// TIA Portal V20 export
DATA_BLOCK "Instance_FB_Recive_Water_Fountain_From_Rework_DB"   // DB105
// stored: AutoNumber false, InstanceOfName FB_Recive_Water_Fountain_From_Rework, InstanceOfType FB
"FB_Recive_Water_Fountain_From_Rework"
   // VAR_INPUT
   //    Emergency_Stop_Release : Bool;
   //    Start : Bool;
   //    Sensor_Water_Fountain_Before_Entrace_Functional_Test_Spinner_Conveyor_Belt : Bool;
   //    Sensor_Water_Fountain_Entrace_Functional_Test_Spinner_Conveyor_Belt : Bool;
   //    Sensor_Spinner_Entrace_Functional_Test_Position_Withdrawn : Bool;
   //    Sensor_Spinner_Entrace_Functional_Test_Position_Advanced : Bool;
   //    Sensor_Water_Fountain_Entrace_Functional_Test_After_Spinner_Conveyor_Belt : Bool;
   //    Sensor_Water_Fountain_Geting_Exit_Rework_Conveyor_Belt : Bool;
   //    Button_Water_Fountain_Get_Exit_Rework_Conveyor_Belt : Bool;
   //    Trigger_Read_Serial_Number_Entrace_Functional_Test : Bool;
   // END_VAR
   // VAR_OUTPUT
   //    Turn_On_Conveyor_Belt_Motor_Spinner_Get_Entrace_Function_Test : Bool;
   //    Valve_Advance_Spinner_Entrace_Functional_Test : Bool;
   //    Signal_Pre_Functional_Test_Production_Line : Bool;
   // END_VAR
   // VAR
   //    Aux_Trig_0 : Bool;
   //    Aux_Trig_1 : Bool;
   //    Aux_Trig_2 : Bool;
   //    Aux_Trig_3 : Bool;
   //    Aux_Trig_4 : Bool;
   //    Aux_Trig_5 : Bool;
   //    Aux_Trig_6 : Bool;
   //    Aux_Trig_7 : Bool;
   //    Aux_Trig_8 : Bool;
   //    Aux_Trig_9 : Bool;
   //    Button_Rework_Pressed : Bool;
   //    "Counter" : USInt;
   //    Timer_Delay_Turn_On_Motor_Spinner_Conveyor_Belt : TON_TIME;
   //    Counter_Water_Fountain_Entrace_Functional_Test { S7_SetPoint := 'True'} : CTUD_USINT;
   // END_VAR
   // VAR RETAIN
   //    Timer_Delay_Spin_Advanced { S7_SetPoint := 'True'} : TON_TIME;
   // END_VAR
   // VAR
   //    Timer_Delay_Spin_Withdrawn { S7_SetPoint := 'True'} : TON_TIME;
   // END_VAR
BEGIN
END_DATA_BLOCK
